{attribute 'GeneratedUsingTerminal: EK1100-0000-0018'}
{attribute addProperty BoxType "EK1100-0000-0018"}
{attribute addProperty Id "Beckhoff_EL7xxxEK1122Beckhoff_EL7xxxEK1122_FF679B322A_0001_EL7031_0000_0016EL7031_AAA74C5945A_0002_EL7031_0000_0017EL7031_AAA74C5945A_0003_EL7031_0000_0018EL7031_022B480446A_0004_EL7031_0000_0019EL7031_022B480446A_0005_EL7031_0000_0020EL7031_022B480446A_0006_EL7031_0000_0021EL7031_022B480446A_0007_EL7031_0000_0022EL7031_022B480446A_0008_EL7031_0000_0023EL7031_022B480446A_0009_EL7031_0000_0024EL7031_022B480446A_0010_EL7031_0000_0025EL7031_022B480446A_0011_EL7031_0000_0026EL7031_022B480446A_0012_EL7031_0030_0016EL7031_B94C493462A_0013_EL7037_0000_0016EL7037_3E4BEAEF54A_0014_EL7037_0000_0017EL7037_3E4BEAEF54A_0015_EL7037_0000_0018EL7037_3E4BEAEF54A_0016_EL7037_0000_0019EL7037_3E4BEAEF54A_0017_EL7037_0000_0020EL7037_3E4BEAEF54A_0018_EL7041_0000_0016EL7041_6D538C6051A_0019_EL7041_0000_0017EL7041_6D538C6051A_0020_EL7041_0000_0018EL7041_C5DF883D52A_0021_EL7041_0000_0019EL7041_C5DF883D52A_0022_EL7041_0000_0020EL7041_C5DF883D52A_0023_EL7041_0000_0021EL7041_C5DF883D52A_0024_EL7041_0000_0022EL7041_C5DF883D52A_0025_EL7041_0000_0023EL7041_C5DF883D52A_0026_EL7041_0000_0024EL7041_C5DF883D52A_0027_EL7041_0000_0025EL7041_C5DF883D52A_0028_EL7041_0001_0016EL7041_B394362F51A_0029_EL7041_0001_0017EL7041_B394362F51A_0030_EL7041_0001_0018EL7041_1B18327252A_0031_EL7041_0001_0019EL7041_1B18327252A_0032_EL7041_0001_0020EL7041_1B18327252A_0033_EL7041_0001_0021EL7041_1B18327252A_0034_EL7041_0001_0022EL7041_1B18327252A_0035_EL7041_0001_0023EL7041_1B18327252A_0036_EL7041_0001_0024EL7041_1B18327252A_0037_EL7041_0052_0016EL7041_022B480446A_0038_EL7041_1000_0016EL7041_6D538C6051A_0039_EL7041_1000_0017EL7041_6D538C6051A_0040_EL7041_1000_0018EL7041_6D538C6051A_0041_EL7041_1000_0019EL7041_6D538C6051A_0042_EL7041_1000_0020EL7041_6D538C6051A_0043_EL7041_1000_0021EL7041_6D538C6051A_0044_EL7047_0000_0016EL7047_3E4BEAEF54A_0045_EL7047_0000_0017EL7047_3E4BEAEF54A_0046_EL7047_0000_0018EL7047_3E4BEAEF54A_0047_EL7047_0000_0019EL7047_3E4BEAEF54A_0048_EL7047_0000_0020EL7047_3E4BEAEF54A_0049_EL7047_0000_0021EL7047_3E4BEAEF54A_0050_EL7047_9014_0021EL7047_3E4BEAEF54A_0051_EL7411_0000_0016EL7411_236AD61B38A_0052_EL7411_0000_0017EL7411_236AD61B38A_0053_EL7411_0000_0018EL7411_236AD61B38"}
{attribute addProperty CRC "2525466581"}
{attribute addProperty Size "2666"}
TYPE Beckhoff_EL7xxx_96878FD5 EXTENDS EK1100_1FC0878B :
STRUCT
	{attribute addProperty Name "Beckhoff_EL7xxxEK1122"}
	{attribute addProperty PreviousPort "Beckhoff EL7xxx : B"}
	Beckhoff_EL7xxxEK1122 : Beckhoff_EL7xxxEK1122_FF679B32;
	{attribute addProperty Name "A_0001_EL7031_0000_0016"}
	{attribute addProperty PreviousPort "Beckhoff EL7xxxEK1122 : C"}
	A_0001_EL7031_0000_0016 : EL7031_AAA74C59;
	{attribute addProperty Name "A_0002_EL7031_0000_0017"}
	{attribute addProperty PreviousPort "A_0001(EL7031-0000-0016) : B"}
	A_0002_EL7031_0000_0017 : EL7031_AAA74C59;
	{attribute addProperty Name "A_0003_EL7031_0000_0018"}
	{attribute addProperty PreviousPort "A_0002(EL7031-0000-0017) : B"}
	A_0003_EL7031_0000_0018 : EL7031_022B4804;
	{attribute addProperty Name "A_0004_EL7031_0000_0019"}
	{attribute addProperty PreviousPort "A_0003(EL7031-0000-0018) : B"}
	A_0004_EL7031_0000_0019 : EL7031_022B4804;
	{attribute addProperty Name "A_0005_EL7031_0000_0020"}
	{attribute addProperty PreviousPort "A_0004(EL7031-0000-0019) : B"}
	A_0005_EL7031_0000_0020 : EL7031_022B4804;
	{attribute addProperty Name "A_0006_EL7031_0000_0021"}
	{attribute addProperty PreviousPort "A_0005(EL7031-0000-0020) : B"}
	A_0006_EL7031_0000_0021 : EL7031_022B4804;
	{attribute addProperty Name "A_0007_EL7031_0000_0022"}
	{attribute addProperty PreviousPort "A_0006(EL7031-0000-0021) : B"}
	A_0007_EL7031_0000_0022 : EL7031_022B4804;
	{attribute addProperty Name "A_0008_EL7031_0000_0023"}
	{attribute addProperty PreviousPort "A_0007(EL7031-0000-0022) : B"}
	A_0008_EL7031_0000_0023 : EL7031_022B4804;
	{attribute addProperty Name "A_0009_EL7031_0000_0024"}
	{attribute addProperty PreviousPort "A_0008(EL7031-0000-0023) : B"}
	A_0009_EL7031_0000_0024 : EL7031_022B4804;
	{attribute addProperty Name "A_0010_EL7031_0000_0025"}
	{attribute addProperty PreviousPort "A_0009(EL7031-0000-0024) : B"}
	A_0010_EL7031_0000_0025 : EL7031_022B4804;
	{attribute addProperty Name "A_0011_EL7031_0000_0026"}
	{attribute addProperty PreviousPort "A_0010(EL7031-0000-0025) : B"}
	A_0011_EL7031_0000_0026 : EL7031_022B4804;
	{attribute addProperty Name "A_0012_EL7031_0030_0016"}
	{attribute addProperty PreviousPort "A_0011(EL7031-0000-0026) : B"}
	A_0012_EL7031_0030_0016 : EL7031_B94C4934;
	{attribute addProperty Name "A_0013_EL7037_0000_0016"}
	{attribute addProperty PreviousPort "A_0012(EL7031-0030-0016) : B"}
	A_0013_EL7037_0000_0016 : EL7037_3E4BEAEF;
	{attribute addProperty Name "A_0014_EL7037_0000_0017"}
	{attribute addProperty PreviousPort "A_0013(EL7037-0000-0016) : B"}
	A_0014_EL7037_0000_0017 : EL7037_3E4BEAEF;
	{attribute addProperty Name "A_0015_EL7037_0000_0018"}
	{attribute addProperty PreviousPort "A_0014(EL7037-0000-0017) : B"}
	A_0015_EL7037_0000_0018 : EL7037_3E4BEAEF;
	{attribute addProperty Name "A_0016_EL7037_0000_0019"}
	{attribute addProperty PreviousPort "A_0015(EL7037-0000-0018) : B"}
	A_0016_EL7037_0000_0019 : EL7037_3E4BEAEF;
	{attribute addProperty Name "A_0017_EL7037_0000_0020"}
	{attribute addProperty PreviousPort "A_0016(EL7037-0000-0019) : B"}
	A_0017_EL7037_0000_0020 : EL7037_3E4BEAEF;
	{attribute addProperty Name "A_0018_EL7041_0000_0016"}
	{attribute addProperty PreviousPort "A_0017(EL7037-0000-0020) : B"}
	A_0018_EL7041_0000_0016 : EL7041_6D538C60;
	{attribute addProperty Name "A_0019_EL7041_0000_0017"}
	{attribute addProperty PreviousPort "A_0018(EL7041-0000-0016) : B"}
	A_0019_EL7041_0000_0017 : EL7041_6D538C60;
	{attribute addProperty Name "A_0020_EL7041_0000_0018"}
	{attribute addProperty PreviousPort "A_0019(EL7041-0000-0017) : B"}
	A_0020_EL7041_0000_0018 : EL7041_C5DF883D;
	{attribute addProperty Name "A_0021_EL7041_0000_0019"}
	{attribute addProperty PreviousPort "A_0020(EL7041-0000-0018) : B"}
	A_0021_EL7041_0000_0019 : EL7041_C5DF883D;
	{attribute addProperty Name "A_0022_EL7041_0000_0020"}
	{attribute addProperty PreviousPort "A_0021(EL7041-0000-0019) : B"}
	A_0022_EL7041_0000_0020 : EL7041_C5DF883D;
	{attribute addProperty Name "A_0023_EL7041_0000_0021"}
	{attribute addProperty PreviousPort "A_0022(EL7041-0000-0020) : B"}
	A_0023_EL7041_0000_0021 : EL7041_C5DF883D;
	{attribute addProperty Name "A_0024_EL7041_0000_0022"}
	{attribute addProperty PreviousPort "A_0023(EL7041-0000-0021) : B"}
	A_0024_EL7041_0000_0022 : EL7041_C5DF883D;
	{attribute addProperty Name "A_0025_EL7041_0000_0023"}
	{attribute addProperty PreviousPort "A_0024(EL7041-0000-0022) : B"}
	A_0025_EL7041_0000_0023 : EL7041_C5DF883D;
	{attribute addProperty Name "A_0026_EL7041_0000_0024"}
	{attribute addProperty PreviousPort "A_0025(EL7041-0000-0023) : B"}
	A_0026_EL7041_0000_0024 : EL7041_C5DF883D;
	{attribute addProperty Name "A_0027_EL7041_0000_0025"}
	{attribute addProperty PreviousPort "A_0026(EL7041-0000-0024) : B"}
	A_0027_EL7041_0000_0025 : EL7041_C5DF883D;
	{attribute addProperty Name "A_0028_EL7041_0001_0016"}
	{attribute addProperty PreviousPort "A_0027(EL7041-0000-0025) : B"}
	A_0028_EL7041_0001_0016 : EL7041_B394362F;
	{attribute addProperty Name "A_0029_EL7041_0001_0017"}
	{attribute addProperty PreviousPort "A_0028(EL7041-0001-0016) : B"}
	A_0029_EL7041_0001_0017 : EL7041_B394362F;
	{attribute addProperty Name "A_0030_EL7041_0001_0018"}
	{attribute addProperty PreviousPort "A_0029(EL7041-0001-0017) : B"}
	A_0030_EL7041_0001_0018 : EL7041_1B183272;
	{attribute addProperty Name "A_0031_EL7041_0001_0019"}
	{attribute addProperty PreviousPort "A_0030(EL7041-0001-0018) : B"}
	A_0031_EL7041_0001_0019 : EL7041_1B183272;
	{attribute addProperty Name "A_0032_EL7041_0001_0020"}
	{attribute addProperty PreviousPort "A_0031(EL7041-0001-0019) : B"}
	A_0032_EL7041_0001_0020 : EL7041_1B183272;
	{attribute addProperty Name "A_0033_EL7041_0001_0021"}
	{attribute addProperty PreviousPort "A_0032(EL7041-0001-0020) : B"}
	A_0033_EL7041_0001_0021 : EL7041_1B183272;
	{attribute addProperty Name "A_0034_EL7041_0001_0022"}
	{attribute addProperty PreviousPort "A_0033(EL7041-0001-0021) : B"}
	A_0034_EL7041_0001_0022 : EL7041_1B183272;
	{attribute addProperty Name "A_0035_EL7041_0001_0023"}
	{attribute addProperty PreviousPort "A_0034(EL7041-0001-0022) : B"}
	A_0035_EL7041_0001_0023 : EL7041_1B183272;
	{attribute addProperty Name "A_0036_EL7041_0001_0024"}
	{attribute addProperty PreviousPort "A_0035(EL7041-0001-0023) : B"}
	A_0036_EL7041_0001_0024 : EL7041_1B183272;
	{attribute addProperty Name "A_0037_EL7041_0052_0016"}
	{attribute addProperty PreviousPort "A_0036(EL7041-0001-0024) : B"}
	A_0037_EL7041_0052_0016 : EL7041_022B4804;
	{attribute addProperty Name "A_0038_EL7041_1000_0016"}
	{attribute addProperty PreviousPort "A_0037(EL7041-0052-0016) : B"}
	A_0038_EL7041_1000_0016 : EL7041_6D538C60;
	{attribute addProperty Name "A_0039_EL7041_1000_0017"}
	{attribute addProperty PreviousPort "A_0038(EL7041-1000-0016) : B"}
	A_0039_EL7041_1000_0017 : EL7041_6D538C60;
	{attribute addProperty Name "A_0040_EL7041_1000_0018"}
	{attribute addProperty PreviousPort "A_0039(EL7041-1000-0017) : B"}
	A_0040_EL7041_1000_0018 : EL7041_6D538C60;
	{attribute addProperty Name "A_0041_EL7041_1000_0019"}
	{attribute addProperty PreviousPort "A_0040(EL7041-1000-0018) : B"}
	A_0041_EL7041_1000_0019 : EL7041_6D538C60;
	{attribute addProperty Name "A_0042_EL7041_1000_0020"}
	{attribute addProperty PreviousPort "A_0041(EL7041-1000-0019) : B"}
	A_0042_EL7041_1000_0020 : EL7041_6D538C60;
	{attribute addProperty Name "A_0043_EL7041_1000_0021"}
	{attribute addProperty PreviousPort "A_0042(EL7041-1000-0020) : B"}
	A_0043_EL7041_1000_0021 : EL7041_6D538C60;
	{attribute addProperty Name "A_0044_EL7047_0000_0016"}
	{attribute addProperty PreviousPort "A_0043(EL7041-1000-0021) : B"}
	A_0044_EL7047_0000_0016 : EL7047_3E4BEAEF;
	{attribute addProperty Name "A_0045_EL7047_0000_0017"}
	{attribute addProperty PreviousPort "A_0044(EL7047-0000-0016) : B"}
	A_0045_EL7047_0000_0017 : EL7047_3E4BEAEF;
	{attribute addProperty Name "A_0046_EL7047_0000_0018"}
	{attribute addProperty PreviousPort "A_0045(EL7047-0000-0017) : B"}
	A_0046_EL7047_0000_0018 : EL7047_3E4BEAEF;
	{attribute addProperty Name "A_0047_EL7047_0000_0019"}
	{attribute addProperty PreviousPort "A_0046(EL7047-0000-0018) : B"}
	A_0047_EL7047_0000_0019 : EL7047_3E4BEAEF;
	{attribute addProperty Name "A_0048_EL7047_0000_0020"}
	{attribute addProperty PreviousPort "A_0047(EL7047-0000-0019) : B"}
	A_0048_EL7047_0000_0020 : EL7047_3E4BEAEF;
	{attribute addProperty Name "A_0049_EL7047_0000_0021"}
	{attribute addProperty PreviousPort "A_0048(EL7047-0000-0020) : B"}
	A_0049_EL7047_0000_0021 : EL7047_3E4BEAEF;
	{attribute addProperty Name "A_0050_EL7047_9014_0021"}
	{attribute addProperty PreviousPort "A_0049(EL7047-0000-0021) : B"}
	A_0050_EL7047_9014_0021 : EL7047_3E4BEAEF;
	{attribute addProperty Name "A_0051_EL7411_0000_0016"}
	{attribute addProperty PreviousPort "A_0050(EL7047-9014-0021) : B"}
	A_0051_EL7411_0000_0016 : EL7411_236AD61B;
	{attribute addProperty Name "A_0052_EL7411_0000_0017"}
	{attribute addProperty PreviousPort "A_0051(EL7411-0000-0016) : B"}
	A_0052_EL7411_0000_0017 : EL7411_236AD61B;
	{attribute addProperty Name "A_0053_EL7411_0000_0018"}
	{attribute addProperty PreviousPort "A_0052(EL7411-0000-0017) : B"}
	A_0053_EL7411_0000_0018 : EL7411_236AD61B;
END_STRUCT
END_TYPE

(* stored: Version 1.2.0.0, ProductVersion 3.1.4024.9
   DUT Beckhoff_EL7xxx_96878FD5: Id {16407538-f3f5-4c37-a2cf-6181513987bd} *)
